TYPE ST_Point :
STRUCT
	X	:LREAL;
	Y	:LREAL;
END_STRUCT
END_TYPE

(* stored: Version 1.1.0.1, ProductVersion 3.1.4026.18
   DUT ST_Point: Id {3c737c80-ac3c-4b6c-a66c-226648dbb8f7} *)
